TYPE Tool_Type :
STRUCT
	speed 				: INT;
	toolNumber 			: INT;
	modelName			: STRING;
	name				: STRING;
END_STRUCT
END_TYPE

(* stored: Version 1.1.0.1, ProductVersion 3.1.4024.12
   DUT Tool_Type: Id {ec2149ba-28e5-4063-89d2-01852d05b58d} *)
